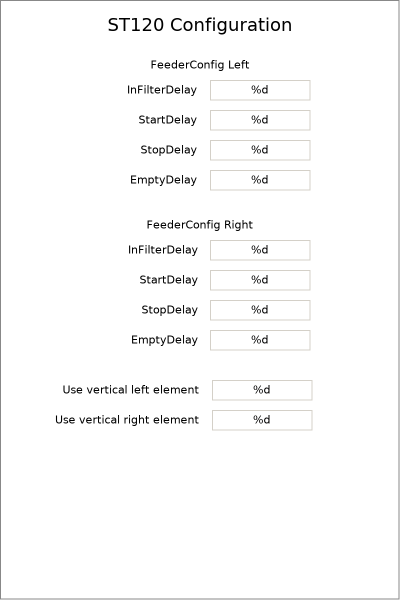
VISUALIZATION VISU_Recipe_ST120  // 400x600
    Textfield (210,80 100x20), "%d", text variable: _20_AUTO.recipe.st120.FeederConfigLeft.InFilterDelay
        OnMouseDown: write the text variable via Default
    Label (0,5 400x40), "ST120 Configuration"
    Label (0,80 200x20), "InFilterDelay"
    Textfield (210,110 100x20), "%d", text variable: _20_AUTO.recipe.st120.FeederConfigLeft.StartDelay
        OnMouseDown: write the text variable via Default
    Label (0,110 200x20), "StartDelay"
    Textfield (210,140 100x20), "%d", text variable: _20_AUTO.recipe.st120.FeederConfigLeft.StopDelay
        OnMouseDown: write the text variable via Default
    Label (0,140 200x20), "StopDelay"
    Textfield (210,170 100x20), "%d", text variable: _20_AUTO.recipe.st120.FeederConfigLeft.EmptyDelay
        OnMouseDown: write the text variable via Default
    Label (0,170 200x20), "EmptyDelay"
    Label (2,380 200x20), "Use vertical left element"
    Label (2,410 200x20), "Use vertical right element"
    Textfield (212,380 100x20), "%d", text variable: _20_AUTO.recipe.st120.xUseVerLeft
        OnMouseDown: write the text variable via Default
    Textfield (212,410 100x20), "%d", text variable: _20_AUTO.recipe.st120.xUseVerRight
        OnMouseDown: write the text variable via Default
    Textfield (210,240 100x20), "%d", text variable: _20_AUTO.recipe.st120.FeederConfigRight.InFilterDelay
        OnMouseDown: write the text variable via Default
    Textfield (210,270 100x20), "%d", text variable: _20_AUTO.recipe.st120.FeederConfigRight.StartDelay
        OnMouseDown: write the text variable via Default
    Textfield (210,300 100x20), "%d", text variable: _20_AUTO.recipe.st120.FeederConfigRight.StopDelay
        OnMouseDown: write the text variable via Default
    Textfield (210,330 100x20), "%d", text variable: _20_AUTO.recipe.st120.FeederConfigRight.EmptyDelay
        OnMouseDown: write the text variable via Default
    Label (100,55 200x20), "FeederConfig Left"
    Label (100,215 200x20), "FeederConfig Right"
    Label (1,240 200x20), "InFilterDelay"
    Label (1,270 200x20), "StartDelay"
    Label (1,300 200x20), "StopDelay"
    Label (1,330 200x20), "EmptyDelay"
END_VISUALIZATION

(* stored: Version 1.1.0.1, ProductVersion 3.1.4024.6
   Visu VISU_Recipe_ST120: Id {ede2f8a6-b1bf-4a0f-bbaf-4f71d489db48} *)
